// TIA Portal project "PlcNetLibrariesS7TestProject" (V14)

(* hardware
DEVICE "S7-1200 station_1"  S7-1200 Station
   slot 0: "Rack_0"  S7-1200 Rack  Rack  V1.0
   slot 1: "PLC_1"  CPU 1212C AC/DC/Rly  6ES7 212-1BE40-0XB0  V4.2
*)

// ===== PLC "PLC_1"  CPU 1212C AC/DC/Rly =====

VAR_GLOBAL   // PLC tag table "Default tag table"
   "TimerReset" AT %M0.1 : Bool;
END_VAR

DATA_BLOCK "Dane"   // DB10
{ S7_Optimized_Access := 'FALSE' }
VERSION : 0.1
   VAR
      Start : Bool;
      Stop : Bool;
      ProcessInProgress : Bool;
      SetPoint : Int := 10;
      CurrentValue : Int;
   END_VAR
BEGIN
END_DATA_BLOCK

// folder: System blocks/Program resources

DATA_BLOCK "Timer1"   // DB1
{ S7_Optimized_Access := 'TRUE' }
AUTHOR : Simatic
FAMILY : IEC
NAME : IEC_TMR
VERSION : 1.0
// stored: InstanceOfName IEC_TIMER
"IEC_TIMER"
BEGIN
END_DATA_BLOCK

// folder: (top level)

ORGANIZATION_BLOCK "Main"   // OB1, LAD, ProgramCycle
TITLE = "Main Program Sweep (Cycle)"
{ S7_Optimized_Access := 'TRUE' }
VERSION : 0.1
   VAR_INPUT
      Initial_Call : Bool;   // Initial call of this OB
      Remanence : Bool;   // =True, if remanent data are available
   END_VAR
   VAR CONSTANT
      ProcessInProgr : Bool;
   END_VAR
BEGIN

REGION Network 1
   // Start handler
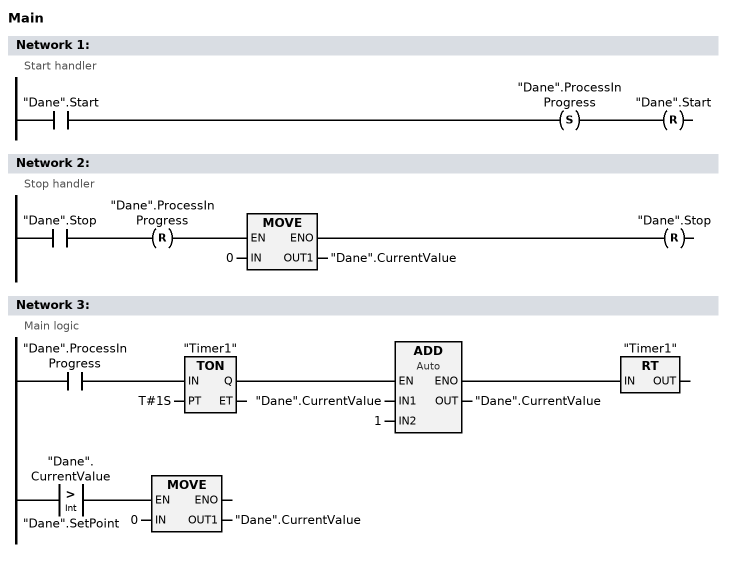
   RUNG wire#powerrail
      Contact( "Dane".Start )
      S_Coil( "Dane".ProcessInProgress )
      R_Coil( "Dane".Start )
   END_RUNG
   // the same network as SCL:
   IF "Dane".Start THEN
       "Dane".ProcessInProgress := TRUE;
       "Dane".Start := FALSE;
   END_IF;
END_REGION

REGION Network 2
   // Stop handler
   RUNG wire#powerrail
      Contact( "Dane".Stop )
      R_Coil( "Dane".ProcessInProgress )
      Move(in := 0, out1 => "Dane".CurrentValue)
      R_Coil( "Dane".Stop )
   END_RUNG
   // the same network as SCL:
   IF "Dane".Stop THEN
       "Dane".ProcessInProgress := FALSE;
       "Dane".CurrentValue := 0;
       "Dane".Stop := FALSE;
   END_IF;
END_REGION

REGION Network 3
   // Main logic
   "Timer1".TON(IN := "Dane".ProcessInProgress, PT := T#1S);
   IF "Timer1".Q THEN
       "Dane".CurrentValue := "Dane".CurrentValue + 1;
       RESET_TIMER("Timer1");
   END_IF;
   IF "Dane".CurrentValue > "Dane".SetPoint THEN "Dane".CurrentValue := 0; END_IF;
END_REGION
END_ORGANIZATION_BLOCK